// SIMATIC STEP 7 (V5.x) project TEMA 5 EJERCICIO 50
// CPU: CPU313 C-2 DP(1)
// station: P_ADR_BUS
// station: Hardware
// station: Equipo SIMATIC 300
// program: Programa S7(1)

SYMBOL_TABLE
"FLANCOS"	DB 1	DB 1
"MANIOBRA"	DB 2	DB 2
"PULSADOR"	I 0.0	BOOL
"FC APERTURA"	I 0.1	BOOL
"FC CIERRE"	I 0.2	BOOL
"Cycle Execution"	OB 1	OB 1
"APERTURA"	Q 0.0	BOOL
"CIERRE"	Q 0.1	BOOL
END_SYMBOL_TABLE

DATA_BLOCK "FLANCOS"	// DB 1
VERSION : 0.1
  STRUCT
   M0 : BOOL ;
   M1 : BOOL ;
   M2 : BOOL ;
   M3 : BOOL ;
   M4 : BOOL ;
   M5 : BOOL ;
   M6 : BOOL ;
   M7 : BOOL ;
   M10 : BOOL ;
   M11 : BOOL ;
   M12 : BOOL ;
   M13 : BOOL ;
   M14 : BOOL ;
   M15 : BOOL ;
   M16 : BOOL ;
   M17 : BOOL ;
   M20 : BOOL ;
   M21 : BOOL ;
   M22 : BOOL ;
   M23 : BOOL ;
   M24 : BOOL ;
   M25 : BOOL ;
   M26 : BOOL ;
   M27 : BOOL ;
  END_STRUCT ;	
BEGIN
END_DATA_BLOCK

DATA_BLOCK "MANIOBRA"	// DB 2
VERSION : 0.1
  STRUCT
   M0 : BOOL ;
   M1 : BOOL ;
   M2 : BOOL ;
   M3 : BOOL ;
   M4 : BOOL ;
   M5 : BOOL ;
   M6 : BOOL ;
   M7 : BOOL ;
   M10 : BOOL ;
   M11 : BOOL ;
   M12 : BOOL ;
   M13 : BOOL ;
   M14 : BOOL ;
   M15 : BOOL ;
  END_STRUCT ;	
BEGIN
END_DATA_BLOCK

ORGANIZATION_BLOCK "Cycle Execution"	// OB 1
TITLE = "Main Program Sweep (Cycle)"
VERSION : 0.1
VAR_TEMP
  OB1_EV_CLASS : BYTE ;	//Bits 0-3 = 1 (Coming event), Bits 4-7 = 1 (Event class 1)
  OB1_SCAN_1 : BYTE ;	//1 (Cold restart scan 1 of OB 1), 3 (Scan 2-n of OB 1)
  OB1_PRIORITY : BYTE ;	//Priority of OB Execution
  OB1_OB_NUMBR : BYTE ;	//1 (Organization block 1, OB1)
  OB1_RESERVED_1 : BYTE ;	//Reserved for system
  OB1_RESERVED_2 : BYTE ;	//Reserved for system
  OB1_PREV_CYCLE : INT ;	//Cycle time of previous OB1 scan (milliseconds)
  OB1_MIN_CYCLE : INT ;	//Minimum cycle time of OB1 (milliseconds)
  OB1_MAX_CYCLE : INT ;	//Maximum cycle time of OB1 (milliseconds)
  OB1_DATE_TIME : DATE_AND_TIME ;	//Date and time OB1 started
END_VAR
BEGIN
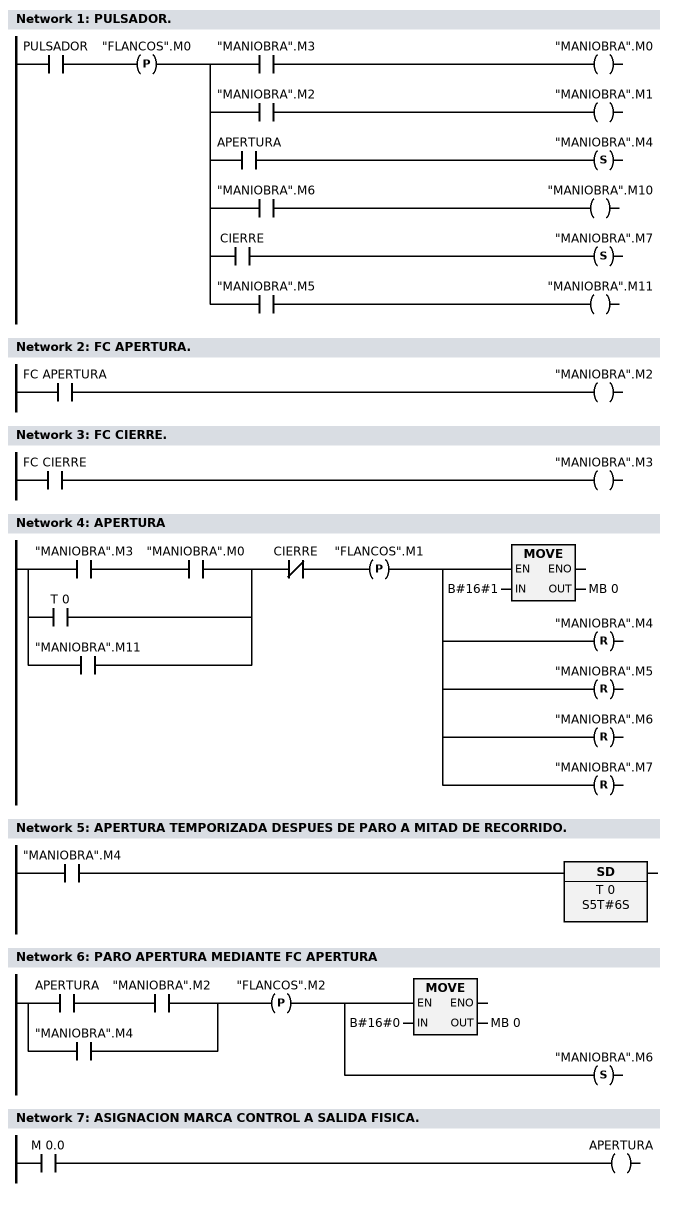
NETWORK
TITLE = PULSADOR.
      A     "PULSADOR";
      FP    "FLANCOS".M0;
      =     L 20.0;
      A     L 20.0;
      A     "MANIOBRA".M3;
      =     "MANIOBRA".M0;
      A     L 20.0;
      A     "MANIOBRA".M2;
      =     "MANIOBRA".M1;
      A     L 20.0;
      A     "APERTURA";
      S     "MANIOBRA".M4;
      A     L 20.0;
      A     "MANIOBRA".M6;
      =     "MANIOBRA".M10;
      A     L 20.0;
      A     "CIERRE";
      S     "MANIOBRA".M7;
      A     L 20.0;
      A     "MANIOBRA".M5;
      =     "MANIOBRA".M11;
NETWORK
TITLE = FC APERTURA.
      A     "FC APERTURA";
      =     "MANIOBRA".M2;
NETWORK
TITLE = FC CIERRE.
      A     "FC CIERRE";
      =     "MANIOBRA".M3;
NETWORK
TITLE = APERTURA 
      A(;
      A     "MANIOBRA".M3;
      A     "MANIOBRA".M0;
      O     T 0;
      O     "MANIOBRA".M11;
      );
      AN    "CIERRE";
      FP    "FLANCOS".M1;
      =     L 20.0;
      A     L 20.0;
      JNB   _001;
      L     B#16#1;
      T     MB 0;
_001: NOP   0;
      A     L 20.0;
      BLD   102;
      R     "MANIOBRA".M4;
      A     L 20.0;
      BLD   102;
      R     "MANIOBRA".M5;
      A     L 20.0;
      BLD   102;
      R     "MANIOBRA".M6;
      A     L 20.0;
      BLD   102;
      R     "MANIOBRA".M7;
NETWORK
TITLE = APERTURA TEMPORIZADA DESPUES DE PARO A MITAD DE RECORRIDO.
      A     "MANIOBRA".M4;
      L     S5T#6S;
      SD    T 0;
NETWORK
TITLE = PARO APERTURA MEDIANTE FC APERTURA
      A(;
      A     "APERTURA";
      A     "MANIOBRA".M2;
      O     "MANIOBRA".M4;
      );
      FP    "FLANCOS".M2;
      =     L 20.0;
      A     L 20.0;
      JNB   _002;
      L     B#16#0;
      T     MB 0;
_002: NOP   0;
      A     L 20.0;
      BLD   102;
      S     "MANIOBRA".M6;
NETWORK
TITLE = ASIGNACION MARCA CONTROL A SALIDA FISICA.
      A     M 0.0;
      =     "APERTURA";
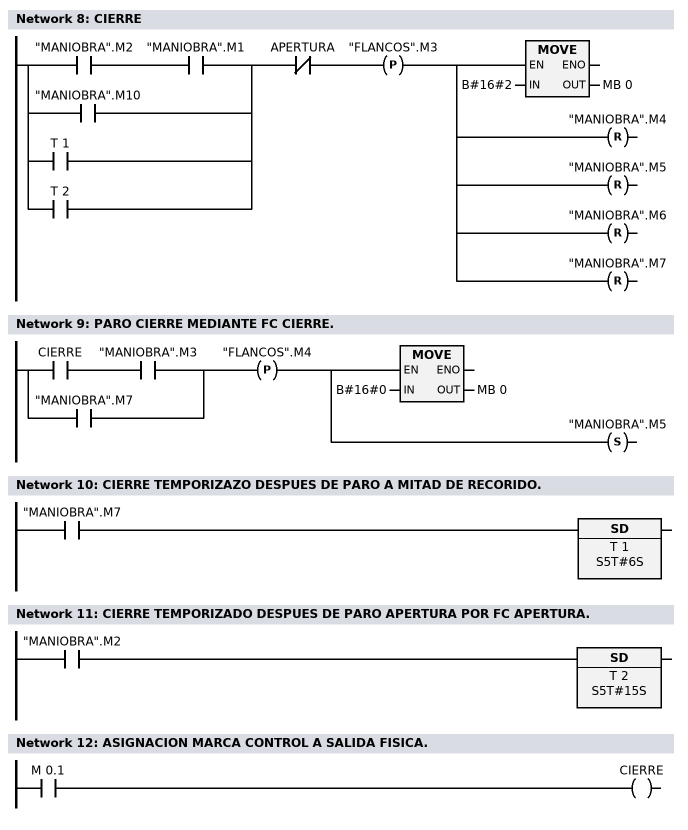
NETWORK
TITLE = CIERRE 
      A(;
      A     "MANIOBRA".M2;
      A     "MANIOBRA".M1;
      O     "MANIOBRA".M10;
      O     T 1;
      O     T 2;
      );
      AN    "APERTURA";
      FP    "FLANCOS".M3;
      =     L 20.0;
      A     L 20.0;
      JNB   _003;
      L     B#16#2;
      T     MB 0;
_003: NOP   0;
      A     L 20.0;
      BLD   102;
      R     "MANIOBRA".M4;
      A     L 20.0;
      BLD   102;
      R     "MANIOBRA".M5;
      A     L 20.0;
      BLD   102;
      R     "MANIOBRA".M6;
      A     L 20.0;
      BLD   102;
      R     "MANIOBRA".M7;
NETWORK
TITLE = PARO CIERRE MEDIANTE FC CIERRE.
      A(;
      A     "CIERRE";
      A     "MANIOBRA".M3;
      O     "MANIOBRA".M7;
      );
      FP    "FLANCOS".M4;
      =     L 20.0;
      A     L 20.0;
      JNB   _004;
      L     B#16#0;
      T     MB 0;
_004: NOP   0;
      A     L 20.0;
      BLD   102;
      S     "MANIOBRA".M5;
NETWORK
TITLE = CIERRE TEMPORIZAZO DESPUES DE PARO A MITAD DE RECORIDO.
      A     "MANIOBRA".M7;
      L     S5T#6S;
      SD    T 1;
NETWORK
TITLE = CIERRE TEMPORIZADO DESPUES DE PARO APERTURA POR FC APERTURA.
      A     "MANIOBRA".M2;
      L     S5T#15S;
      SD    T 2;
NETWORK
TITLE = ASIGNACION MARCA CONTROL A SALIDA FISICA.
      A     M 0.1;
      =     "CIERRE";
END_ORGANIZATION_BLOCK
